Staubli VAL3: lower.pgx

public program lower(string& sText)
  local num i
  local num n
begin
  // Converts all lowercase letter of a string to uppercase
  //
  // copyright (c) 2017-2021 victortorreslopez
  //
  // GNU General Public License
  //
  // Parameters
  // - &sText: source string
  //
  // Local variables
  // - i: iterator index
  // - n: current char unicode code
  //
  // Version history
  // ---------------
  // 0.0, 2021/12/21, VTL: 1st update (coding style)
  // 0.0, 2017/01/04, VTL: alfa release

  for i = 0 to len(sText) - 1
    n = asc(sText, i)
    if (n > 65) and (n < 90)
      sText = replace(sText, chr(n + 32), 1, i)
    endIf
  endFor
end
